FUNCTION_BLOCK FB_FormingBoardControl_V3

VAR_INPUT

    //────────────────────────────────────────────
    // GROUP / INTERLOCKS
    //────────────────────────────────────────────
    startGroup              : BOOL; // Start command (pulse) / Comando de partida (pulso)
    stopGroup               : BOOL; // Stop command (level) / Comando de parada (nível)
    fastStopGroup               : BOOL; // Stop command (level) / Comando de parada (nível)
	groupReset              : BOOL; // Fault reset / Reset de falhas do grupo
	
    //────────────────────────────────────────────
    // AUXILIARY MOTORS — INDICATORS & COMMANDS
    //────────────────────────────────────────────
    grouSpeedDifIncCmd      : BOOL; // Lamp: offset increasing / Lâmpada: aumento de offset
    grouSpeedDifDecCmd      : BOOL; // Lamp: offset decreasing / Lâmpada: redução de offset
	
    //────────────────────────────────────────────
    // SPEED ADJUSTMENTS / OFFSET TUNING
    //────────────────────────────────────────────
    groupRecoverSpeedCmd    : BOOL; // Recover speed while TRUE / Recuperar velocidade enquanto TRUE
    //────────────────────────────────────────────
    // DRIVE STATUS INPUTS — FORMING BOARD ROLLS
    //────────────────────────────────────────────
    tractionRollReady       : BOOL; // MASTER ready / Pronto (mestre)
    suctionRollReady        : BOOL; // SLAVE ready / Pronto (seguidor)
	paperPresenceSensor : BOOL;

    //────────────────────────────────────────────
    // SPEED SETPOINTS / MODE
    //────────────────────────────────────────────
    groupAutoSpeedMPM       : REAL;       // Auto mode speed [m/min]
    groupManualSpeedMPM     : REAL := 50.0; // Manual mode speed
    groupSpeedAutoMan       : BOOL;       // 0=Manual, 1=Auto

    //────────────────────────────────────────────
    // SPEED & TORQUE FEEDBACKS
    //────────────────────────────────────────────
    tractionRollSpeedFeedback     : REAL; // MASTER speed feedback
    tractionRollTorqueFeedback    : REAL; // MASTER torque feedback
    suctionRollSpeedFeedback      : REAL; // SLAVE speed feedback
    suctionRollTorqueFeedback     : REAL; // SLAVE torque feedback

    //────────────────────────────────────────────
    // WIRE/FELT EDGE / RUNNING SAFETY SENSORS
    //────────────────────────────────────────────
    formingBoardWireOverrunSensorOperatorSide : BOOL; // Operator side / Lado operador
    formingBoardWireOverrunSensorDriveSide    : BOOL; // Drive side / Lado comando

    machineConfig : PaperMachine_TypeHmiConfig;

END_VAR



VAR_OUTPUT

    //────────────────────────────────────────────
    // STATE / DIAGNOSTICS
    //────────────────────────────────────────────
    deviceState                 : STRING; // Current state string / Estado atual em texto
    statusCode                  : INT;    // 0=Idle, 1=Starting, 2=Running, 3=Fault
    groupFault                  : BOOL;   // TRUE if any group fault active / Falha geral do grupo
	speedDifError: BOOL;

    //────────────────────────────────────────────
    // SPEED REFERENCES (TO DRIVES) AND DISPLAY
    //────────────────────────────────────────────
    tractionRollSpeedSetpointRPM : REAL; // MASTER speed reference [rpm]
    suctionRollSpeedSetpointRPM  : REAL; // SLAVE speed reference [rpm]

    tractionRollSpeedFeedbackRPM : REAL; // MASTER speed feedback [rpm]
    suctionRollSpeedFeedbackRPM  : REAL; // SLAVE speed feedback [rpm]

    tractionRollSpeedFeedbackMPM : REAL; // MASTER speed feedback [m/min]
    suctionRollSpeedFeedbackMPM  : REAL; // SLAVE speed feedback [m/min]

    tractionRollTorqueFeedbackPct : REAL; // MASTER torque feedback [%]
    suctionRollTorqueFeedbackPct  : REAL; // SLAVE torque feedback [%]

    nextGroupSpeedRefMPM        : REAL; // Next group speed [m/min]

    //────────────────────────────────────────────
    // TORQUE REFERENCES / LIMITS (SLAVE)
    //────────────────────────────────────────────
    suctionRollTorqueRefPct     : REAL; // Torque setpoint for SLAVE [%]

    //────────────────────────────────────────────
    // DRIVE COMMANDS (ENABLE / RESET)
    //────────────────────────────────────────────
    tractionRollDriveEnable     : BOOL; // Enable MASTER drive
    tractionRollDriveReset      : BOOL; // Reset MASTER drive fault
    suctionRollDriveEnable      : BOOL; // Enable SLAVE drive
    suctionRollDriveReset       : BOOL; // Reset SLAVE drive fault

    //────────────────────────────────────────────
    // STATUS CODES (PER DRIVE)
    //────────────────────────────────────────────


    //────────────────────────────────────────────
    // HMI ALARMS STRUCTURE
    //────────────────────────────────────────────
    hmiAlarms                   : PaperMachine_TypeHmiAlarms;

END_VAR



VAR
    instFB_GroupDriveControl_V1       : FB_GroupDriveControl_V1;
    instFB_GroupSpeedControl_V1       : FB_GroupSpeedControl_V1;
	instFB_FormingBoardSpeedControl	: FB_FormingBoardSpeedControl;
    instFB_GroupDisplayFilters_V1     : FB_GroupDisplayFilters_V1;
    instFB_GroupTorqueTrimControl_V1  : FB_GroupTorqueTrimControl_V1;
	
	instFB_GroupTorqueTrimControl_V2  : FB_GroupTorqueTrimControl_V2;

	speedDif: REAL;
	instTONWireOverRunTrip: TON;
	instTONSpeedDifDelay: TON;
	instTOF_PaperPresenseDelay : TOF;	
	
	instTPSpeedDifErrorHold: TP;
END_VAR

VAR PERSISTENT
END_VAR

// ─────────────────────────────────────────────────────────────────────────────
// MAIN CALL SEQUENCE
// ─────────────────────────────────────────────────────────────────────────────

_GroupControl();          // 1) State machine: edges, enables, stop modes
_StateDisplay();
_SpeedDifferenceCheck();  // 4) Speed difference monitor & trip
_auxiliaryControls();

_alarmsDisplay();

METHOD _alarmsDisplay
VAR_INPUT
END_VAR
(*
//==============================================================
// FAULT EVALUATION — PER CONDITION (flags only; no global set)
//==============================================================

//----------------------------
// PRESS SECTION DRIVES
//----------------------------
hmiAlarms.pressSectionFirstPressFaultAlarm  := firstPressVfdFaultFeedback;
hmiAlarms.pressSectionSecondPressFaultAlarm := secondPressVfdFaultFeedback;

//----------------------------
// PRESS SECTION AUXILIARIES
//----------------------------
hmiAlarms.pressSectionUpperFeltStretcherFaultAlarm := upperFelt1StretcherFault;
hmiAlarms.pressSectionLowerFeltStretcherFaultAlarm := lowerFeltStretcherFault;
hmiAlarms.pressSectionUpperInfeedRollFaultAlarm    := upperInfeedRollFault;
hmiAlarms.pressSectionLowerInfeedRollFaultAlarm    := lowerInfeedRollFault;


//==============================================================
// PRESS SECTION — FELT EDGE OVERRUN ALARMS (DIRECT SENSORS)
//==============================================================

hmiAlarms.pressSectionUpperFelt1OverrunOperatorSideAlarm := pressSectionUpperFelt1OverrunSensorOperatorSide;
hmiAlarms.pressSectionUpperFelt1OverrunDriveSideAlarm    := pressSectionUpperFelt1OverrunSensorDriveSide;

hmiAlarms.pressSectionUpperFelt2OverrunOperatorSideAlarm := pressSectionUpperFelt2OverrunSensorOperatorSide;
hmiAlarms.pressSectionUpperFelt2OverrunDriveSideAlarm    := pressSectionUpperFelt2OverrunSensorDriveSide;

hmiAlarms.pressSectionLowerFeltOverrunOperatorSideAlarm := pressSectionLowerFeltOverrunSensorOperatorSide;
hmiAlarms.pressSectionLowerFeltOverrunDriveSideAlarm    := pressSectionLowerFeltOverrunSensorDriveSide;


//----------------------------
// PRESS SECTION GROUP FAULT STATUS
//----------------------------
groupFault :=
    hmiAlarms.pressSectionFirstPressFaultAlarm 
	OR hmiAlarms.pressSectionSecondPressFaultAlarm 
	OR hmiAlarms.pressFelt1OverrunOperatorSideAlarm
	OR hmiAlarms.pressFelt1OverrunDriveSideAlarm
	OR hmiAlarms.pressFelt2OverrunOperatorSideAlarm
	OR hmiAlarms.pressFelt2OverrunDriveSideAlarm
	OR hmiAlarms.pressFelt3OverrunOperatorSideAlarm
	OR hmiAlarms.pressFelt3OverrunDriveSideAlarm;


*)
//==============================================================
// FAULT EVALUATION — PER CONDITION (flags only; no global set)
//==============================================================

//----------------------------
// PRESS SECTION DRIVES
//----------------------------
//hmiAlarms.pressSectionFirstPressFaultAlarm  := firstPressVfdFaultFeedback;
//hmiAlarms.pressSectionSecondPressFaultAlarm := secondPressVfdFaultFeedback;

//----------------------------
// PRESS SECTION AUXILIARIES
//----------------------------
END_METHOD

METHOD _auxiliaryControls
VAR_INPUT
END_VAR
END_METHOD

METHOD _GroupControl
VAR_INPUT
END_VAR


(*
    formingBoardTorquePIDCtrlKp                   : REAL := 2.0;
    formingBoardTorquePIDCtrlTn                   : REAL := 8.0;
    formingBoardTorquePIDCtrlTv                   : REAL := 0.0;
    formingBoardTorqueLimit                   : REAL := 100.0;
	
*)
VAR
	suctionRollTorqueRefPct_: REAL;
END_VAR
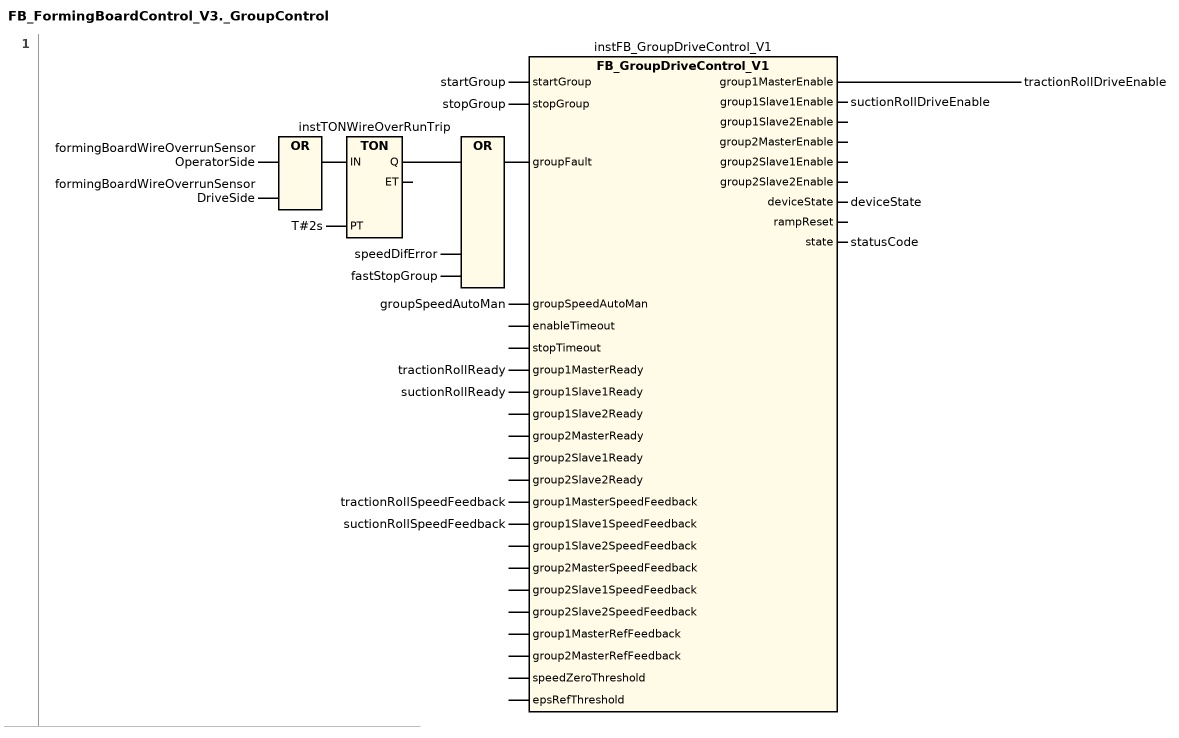
// NETWORK 1
instTONWireOverRunTrip(IN := formingBoardWireOverrunSensorOperatorSide OR formingBoardWireOverrunSensorDriveSide, PT := T#2s); // TON
instFB_GroupDriveControl_V1(
    startGroup := startGroup,
    stopGroup := stopGroup,
    groupFault := instTONWireOverRunTrip.Q OR speedDifError OR fastStopGroup,
    groupSpeedAutoMan := groupSpeedAutoMan,
    group1MasterReady := tractionRollReady,
    group1Slave1Ready := suctionRollReady,
    group1MasterSpeedFeedback := tractionRollSpeedFeedback,
    group1Slave1SpeedFeedback := suctionRollSpeedFeedback,
    group1Slave1Enable => suctionRollDriveEnable,
    deviceState => deviceState,
    state => statusCode); // FB_GroupDriveControl_V1
tractionRollDriveEnable := instFB_GroupDriveControl_V1.group1MasterEnable;

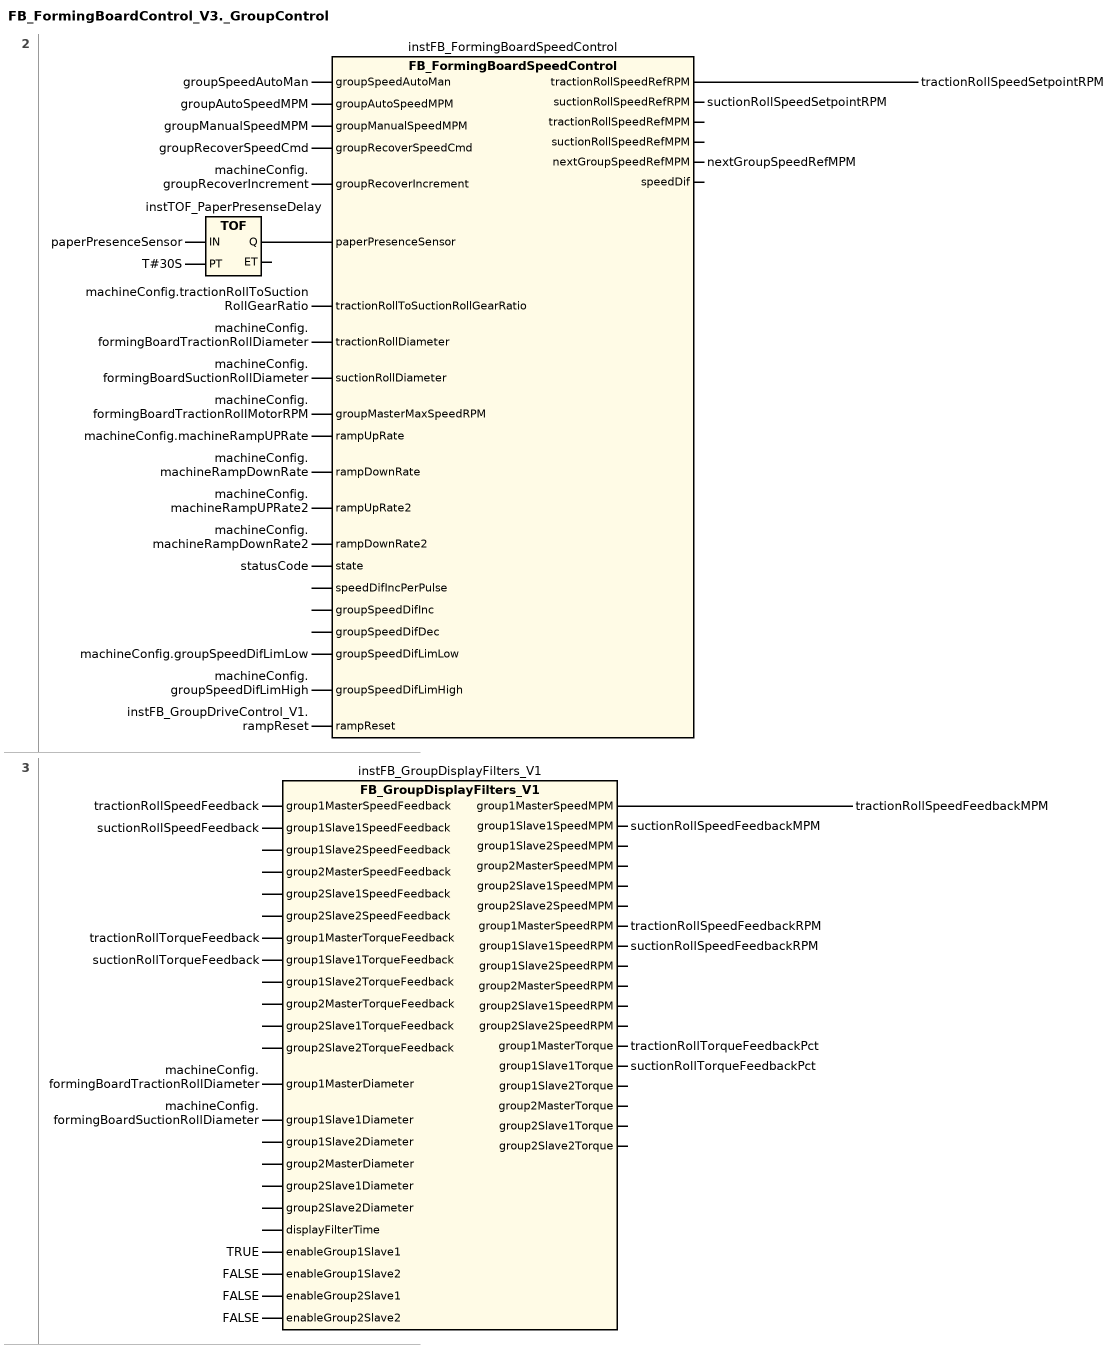
// NETWORK 2
instTOF_PaperPresenseDelay(IN := paperPresenceSensor, PT := T#30S); // TOF
instFB_FormingBoardSpeedControl(
    groupSpeedAutoMan := groupSpeedAutoMan,
    groupAutoSpeedMPM := groupAutoSpeedMPM,
    groupManualSpeedMPM := groupManualSpeedMPM,
    groupRecoverSpeedCmd := groupRecoverSpeedCmd,
    groupRecoverIncrement := machineConfig.groupRecoverIncrement,
    paperPresenceSensor := instTOF_PaperPresenseDelay.Q,
    tractionRollToSuctionRollGearRatio := machineConfig.tractionRollToSuctionRollGearRatio,
    tractionRollDiameter := machineConfig.formingBoardTractionRollDiameter,
    suctionRollDiameter := machineConfig.formingBoardSuctionRollDiameter,
    groupMasterMaxSpeedRPM := machineConfig.formingBoardTractionRollMotorRPM,
    rampUpRate := machineConfig.machineRampUPRate,
    rampDownRate := machineConfig.machineRampDownRate,
    rampUpRate2 := machineConfig.machineRampUPRate2,
    rampDownRate2 := machineConfig.machineRampDownRate2,
    state := statusCode,
    groupSpeedDifLimLow := machineConfig.groupSpeedDifLimLow,
    groupSpeedDifLimHigh := machineConfig.groupSpeedDifLimHigh,
    rampReset := instFB_GroupDriveControl_V1.rampReset,
    suctionRollSpeedRefRPM => suctionRollSpeedSetpointRPM,
    nextGroupSpeedRefMPM => nextGroupSpeedRefMPM); // FB_FormingBoardSpeedControl
tractionRollSpeedSetpointRPM := instFB_FormingBoardSpeedControl.tractionRollSpeedRefRPM;

// NETWORK 3
instFB_GroupDisplayFilters_V1(
    group1MasterSpeedFeedback := tractionRollSpeedFeedback,
    group1Slave1SpeedFeedback := suctionRollSpeedFeedback,
    group1MasterTorqueFeedback := tractionRollTorqueFeedback,
    group1Slave1TorqueFeedback := suctionRollTorqueFeedback,
    group1MasterDiameter := machineConfig.formingBoardTractionRollDiameter,
    group1Slave1Diameter := machineConfig.formingBoardSuctionRollDiameter,
    enableGroup1Slave1 := TRUE,
    enableGroup1Slave2 := FALSE,
    enableGroup2Slave1 := FALSE,
    enableGroup2Slave2 := FALSE,
    group1Slave1SpeedMPM => suctionRollSpeedFeedbackMPM,
    group1MasterSpeedRPM => tractionRollSpeedFeedbackRPM,
    group1Slave1SpeedRPM => suctionRollSpeedFeedbackRPM,
    group1MasterTorque => tractionRollTorqueFeedbackPct,
    group1Slave1Torque => suctionRollTorqueFeedbackPct); // FB_GroupDisplayFilters_V1
tractionRollSpeedFeedbackMPM := instFB_GroupDisplayFilters_V1.group1MasterSpeedMPM;

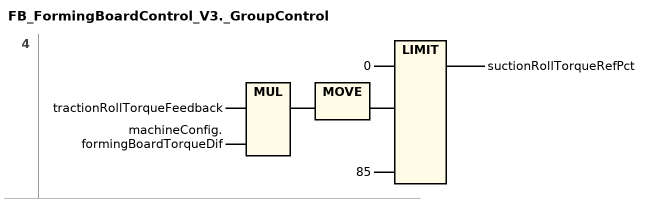
// NETWORK 4
suctionRollTorqueRefPct := LIMIT(0, tractionRollTorqueFeedback * machineConfig.formingBoardTorqueDif, 85);
END_METHOD

METHOD PRIVATE _Scale : REAL
VAR_INPUT
    X    : REAL;
    I_LO : REAL;
    I_HI : REAL;
    O_LO : REAL;
    O_HI : REAL;
END_VAR
IF I_LO = I_HI THEN
	_Scale := O_LO;
ELSE
	_Scale := (O_HI - O_LO) / (I_HI - I_LO) * (LIMIT(I_LO, X, I_HI) - I_LO) + O_LO;
END_IF;
END_METHOD

// ============================== Methods ==============================
// Intra-section speed supervision for Press Section (firstPress ↔ secondPress)
METHOD _SpeedDifferenceCheck
(*

    tractionRollSpeedFeedbackMPM : REAL; // MASTER speed feedback [m/min]
    suctionRollSpeedFeedbackMPM  : REAL; // SLAVE speed feedback [m/min]

*)
speedDif := ABS(tractionRollSpeedFeedbackMPM - suctionRollSpeedFeedbackMPM);


// Timer de confirmação do erro
instTONSpeedDifDelay(
    IN := speedDif > 50,
    PT := T#3S
);


// Pulso para segurar o status do erro por 100 ms
instTPSpeedDifErrorHold(
    IN := instTONSpeedDifDelay.Q,
    PT := T#100MS
);


// Status final do erro
speedDifError := instTPSpeedDifErrorHold.Q;
END_METHOD

METHOD _StateDisplay
VAR_INPUT
END_VAR

// ──────────────────────────────────────────────────────────────────────────────
// _StateDisplay — Press Section (firstPress = Master, secondPress = Slave)
// Maps the internal machine "state" to a compact HMI status code and derives
// per-drive motor status codes from VFD signals.
//
// statusCode / firstPressStatusCode / secondPressStatusCode legend:
//   0 = Idle, 1 = Starting, 2 = Running, 3 = Fault
//
// Machine "state" groups:
//   0 = IDLE, 1 = ENABLE, 2 = WAIT_EN, 3 = RAMP_EN, 4 = RUN, 5 = STOPPING, 10 = FAULT
// Priority rule (for motors): Fault > Running > Starting > Idle
// ──────────────────────────────────────────────────────────────────────────────
VAR CONSTANT
    STATUS_IDLE     : INT := 0;
    STATUS_STARTING : INT := 1;
    STATUS_RUNNING  : INT := 2;
    STATUS_FAULT    : INT := 3;
END_VAR
END_METHOD

END_FUNCTION_BLOCK

(* stored: Version 1.1.0.1, ProductVersion 3.1.4024.15
   POU FB_FormingBoardControl_V3: Id {43ced332-d776-436e-a89d-0a538917f1bf}, SpecialFunc None
   Method _alarmsDisplay: Id {b9c8e0e7-09b4-4c30-bdc0-74f665aa3b30}
   Method _auxiliaryControls: Id {c83736e7-eaa4-4314-98af-c1e4d9b768b8}
   Method _GroupControl: Id {9e47b46c-970e-4d76-953c-b5028d61d2a5}
   Method _Scale: Id {d272cee9-8d42-4951-b59a-a0a5b87266ed}
   Method _SpeedDifferenceCheck: Id {517346dd-3710-4c3a-b13d-3a526144ca07}
   Method _StateDisplay: Id {c51260d8-b357-494a-859d-3b8c07339490} *)
